{attribute 'qualified_only'}
VAR_GLOBAL
	vaerde: INT;
	
END_VAR

(* stored: Version 1.1.0.1, ProductVersion 3.1.4024.11
   GVL GVL: Id {3738c192-e713-4209-a6f3-4ca47426ed9e} *)
